Staubli VAL3: Binary7En.dtx

bool bRead
public mdesc mNomSpeed
num nKey
string sBit[16] = "1010011010"
string sMenu[8]
  [2] = "F1: Decimal (num) to Binary (string)"
  [3] = "F2: Binary (string) to Decimal (num)"
  [4] = "F3: Operator function"
  [5] = "F4: Power calculation"
  [6] = "F5: And function (num and num)"
  [7] = "F6: Write 16 bit word"
string sSubMenu[7]
  [2] = "F1: And function"
  [3] = "F2: Or function"
  [4] = "F3: Xor function"
  [5] = "F4: Nand function"
  [6] = "F5: Nor function"
string sDec2HexSymbols[16]
  [0] = "0"
  [1] = "1"
  [2] = "2"
  [3] = "3"
  [4] = "4"
  [5] = "5"
  [6] = "6"
  [7] = "7"
  [8] = "8"
  [9] = "9"
  [10] = "A"
  [11] = "B"
  [12] = "C"
  [13] = "D"
  [14] = "E"
  [15] = "F"
string sDecHexBuff
string sHexDecBuff
num nHex2DecSymbols{}
  [0] = {}
  [1] = 1
  [8] = 8
  [9] = 9
  [A] = 10
  [B] = 11
  [C] = 12
  [D] = 13
  [E] = 14
  [F] = 15
  [2] = 2
  [3] = 3
  [4] = 4
  [5] = 5
  [6] = 6
  [7] = 7
